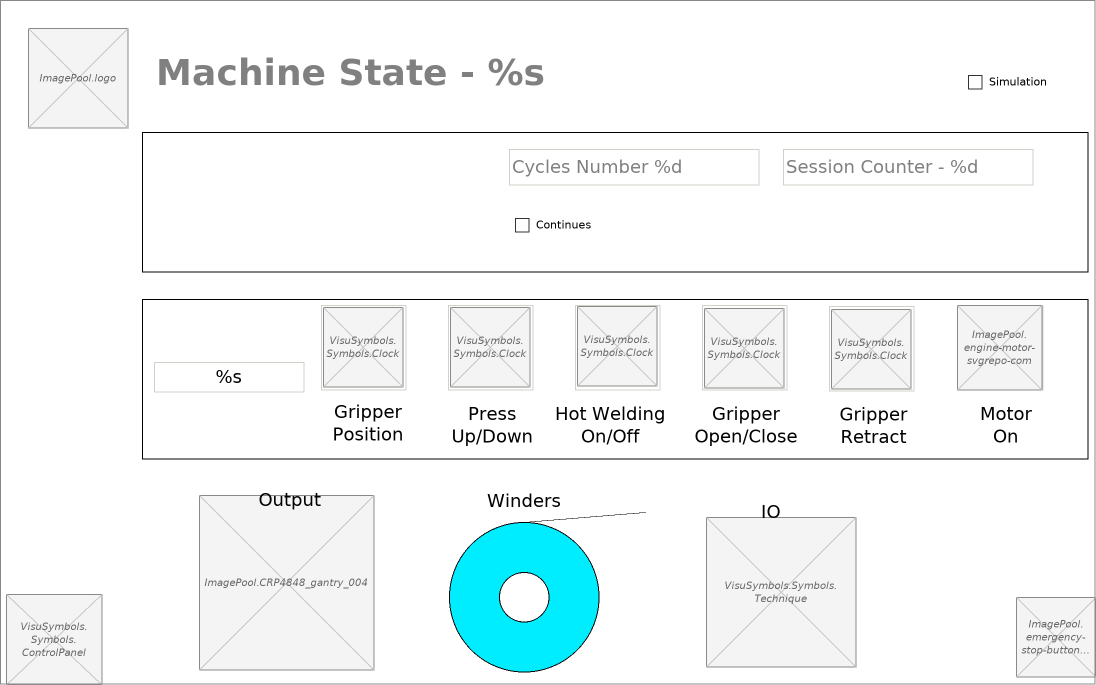
VISUALIZATION Visualization  // 1096x685
    RoundedRectangle (142,299 946x160)
    RoundedRectangle (142,132 946x140)
    Image (28,28 100x100), image: ImagePool.logo
        p2858320360: HMI.LogoRotation
    RoundedRectangle (267,147 100x100), colour toggle: HMI.StartButtonColor
    Image (278,159 75x75), image: ImagePool.play-button-svgrepo-com
    RoundedRectangle (268,147 100x100)
        tap gMachineCtrl.Cmd.Start
        OnMouseEnter: toggle HMI.StartButtonColor
        OnMouseLeave: toggle HMI.StartButtonColor
    Group (378,147 100x100)
        RoundedRectangle (0,0 100x100), colour toggle: HMI.StopButtonColor
        Image (14,12 75x75), image: ImagePool.stop-svgrepo-com
        RoundedRectangle (0,0 100x100)
            tap gMachineCtrl.Cmd.Stop
            OnMouseEnter: toggle HMI.StopButtonColor
            OnMouseLeave: toggle HMI.StopButtonColor
    Textfield (153,41 743x63), "Machine State - %s", text variable: FB_Machine_Ctrl.Monitoring.StepMessage
    Checkbox (513,205 150x40), "Continues", variable: gMachineCtrl.Parameters.Continues
    Textfield (509,149 250x36), "Cycles Number %d", text variable: gMachineCtrl.Parameters.NumberOfCycles, input disabled if: gMachineCtrl.Parameters.Continues
        OnMouseClick: write the text variable via Edit, min 0, max 1000000, title "Enter number of cycles"
    Textfield (783,149 250x36), "Session Counter - %d", text variable: gMachineCtrl.Status.SessionCounter
    Textfield (154,362 150x30), "%s", text variable: FB_Machine_Run.Delay.ET
    RoundedRectangle (321,305 85x85), colour toggle: HMI.TimerGripperPostionColor
    Image (323,307 80x80), image: VisuSymbols.Symbols.Clock
        OnMouseClick: OpenDialog Dialog=DialogTimer_GripperPosi, OpenModal=True, OpenCentered=True
    Label (313,389 110x68), "Gripper Position"
    Label (549,393 123x64), "Hot Welding On/Off"
    Label (685,395 122x60), "Gripper Open/Close"
    Label (824,397 99x57), "Gripper Retract"
    Label (443,386 99x78), "Press Up/Down"
    RoundedRectangle (448,305 85x85), colour toggle: HMI.TimerHotWeldColor
    Image (450,307 80x80), image: VisuSymbols.Symbols.Clock
        OnMouseClick: OpenDialog Dialog=DialogTimer_HotWeldValve, OpenModal=True, OpenCentered=True
    RoundedRectangle (575,305 85x85), colour toggle: HMI.TimerHeaterOnColor
    Image (577,306 80x80), image: VisuSymbols.Symbols.Clock
        OnMouseClick: OpenDialog Dialog=DialogTimer_HeaterOn, OpenModal=True, OpenCentered=True
    RoundedRectangle (702,305 85x85), colour toggle: HMI.TimerGripperopenColor
    Image (704,308 80x80), image: VisuSymbols.Symbols.Clock
        OnMouseClick: OpenDialog Dialog=DialogTimer_GripperOpenClose, OpenModal=True, OpenCentered=True
    RoundedRectangle (829,306 85x85), colour toggle: HMI.TimerGripperRetractColor
    Image (831,309 80x80), image: VisuSymbols.Symbols.Clock
        OnMouseClick: OpenDialog Dialog=DialogTimer_ValveClose, OpenModal=True, OpenCentered=True
    RoundedRectangle (958,305 85x85), colour toggle: HMI.StateMotorOnColor
    Label (972,391 68x68), "Motor On"
    Image (957,305 85x85), image: ImagePool.engine-motor-svgrepo-com
    Image (1016,597 80x80), image: ImagePool.emergency-stop-button-icon-364856
        p1097714728: HMI.EstopScalling
        OnMouseClick: toggle gMachineCtrl.Cmd.EmStop
        OnMouseDown: execute { HMI.EstopScalling	:= 1100; }
        OnMouseUp: execute { HMI.EstopScalling	:= 1300; }
        OnMouseEnter: execute { HMI.EstopScalling	:= 1300; }
        OnMouseLeave: execute { HMI.EstopScalling	:= 1000; }
    Checkbox (966,67 109x30), "Simulation", variable: gMachineCtrl.Simulation
    RoundedRectangle (166,151 100x100), colour toggle: HMI.SwitchOnButtonColor
    Image (185,163 64x64), image: ImagePool.power-power-button-svgrepo-com
        p1097714728: HMI.onOffScaling
    RoundedRectangle (165,150 100x100)
        toggle gMachineCtrl.Cmd.SwitchOn
        OnMouseEnter: execute { HMI.SwitchOnButtonColor :=TRUE; HMI.onOffScaling		:=1200; }
        OnMouseLeave: execute {
            IF gMachineCtrl.Cmd.SwitchOn THEN
            	HMI.SwitchOnButtonColor:=TRUE;
            ELSE
            	HMI.SwitchOnButtonColor:=FALSE;
            END_IF
            HMI.onOffScaling		:=1000;
        }
    Group (449,486 196x186)
        p1097714728: HMI.WinderScaling
        OnMouseClick: OpenDialog Dialog=Winders, OpenModal=True, OpenCentered=True
        OnDialogClosed: execute { HMI.WinderScaling := 1000; }
        OnMouseDown: execute { HMI.WinderScaling := 1000; }
        OnMouseEnter: execute { HMI.WinderScaling := 1100; }
        OnMouseLeave: execute { HMI.WinderScaling := 1000; }
        Label (0,0 150x30), "Winders"
        Ellipse (0,36 150x150)
            OnMouseDown: OpenDialog Dialog=Winders, OpenModal=True, OpenCentered=True
        Ellipse (50,86 50x50)
        Line (62,37) (196,26)
    Image (6,594 96x91), image: VisuSymbols.Symbols.ControlPanel
        p1097714728: HMI.SettingsScaling
        OnMouseClick: OpenDialog Dialog=Dialog_Settings, OpenModal=True, OpenCentered=True
        OnDialogClosed: execute { HMI.SettingsScaling:=1000; }
        OnMouseDown: execute { HMI.SettingsScaling:=1000; }
        OnMouseEnter: execute { HMI.SettingsScaling:=1100; }
        OnMouseLeave: execute { HMI.SettingsScaling:=1000; }
    Group (696,497 160x170)
        p1097714728: HMI.IOScaling
        OnMouseClick: OpenDialog Dialog=Dialog_IO, OpenModal=True, OpenCentered=True
        OnMouseLeave: execute { HMI.IOScaling:=1000; }
        OnDialogClosed: execute { HMI.IOScaling:=1000; }
        OnMouseEnter: execute { HMI.IOScaling:=1150; }
        Image (10,20 150x150), image: VisuSymbols.Symbols.Technique
            OnMouseClick: OpenDialog Dialog=Dialog_IO, OpenModal=True, OpenCentered=True
        Label (0,0 150x30), "IO"
    Image (199,495 175x175), image: ImagePool.CRP4848_gantry_004
        p1097714728: HMI.OutputScaling
        OnMouseClick: OpenDialog Dialog=Dialog_Output, OpenModal=True, OpenCentered=True
        OnMouseDown: execute { HMI.OutputScaling:=1000; }
        OnDialogClosed: execute { HMI.OutputScaling:=1000; }
        OnMouseLeave: execute { HMI.OutputScaling:=1000; }
        OnMouseEnter: execute { HMI.OutputScaling:=1100; }
    Label (215,485 150x30), "Output"
END_VISUALIZATION

(* stored: Version 1.1.0.1, ProductVersion 3.1.4024.3
   Visu Visualization: Id {c720a588-1e5f-4d94-aeb1-f1463c06cc1a} *)
